//tcUNIT Common function block: Contains helper methods for tcUNIT.
FUNCTION_BLOCK FB_tcUNIT_common

VAR

END_VAR

METHOD mDisableAxis: BOOL
VAR_INPUT
    iAxisIndex: UINT; //The idex of the axis to action the method on.
END_VAR
GVL.astAxes[iAxisIndex].stControl.bEnable := FALSE;
END_METHOD

METHOD mEnableAxis: BOOL
VAR_INPUT
    iAxisIndex: UINT; //The idex of the axis to action the method on.
END_VAR
GVL.astAxes[iAxisIndex].stControl.bEnable := TRUE;
END_METHOD

METHOD mExecute: BOOL
VAR_INPUT
    iAxisIndex: UINT; //The idex of the axis to action the method on.
END_VAR
GVL.astAxes[iAxisIndex].stControl.bExecute := TRUE;
END_METHOD

METHOD mExecute_SetFALSE: BOOL
VAR_INPUT
    iAxisIndex: UINT; //The idex of the axis to action the method on.
END_VAR
GVL.astAxes[iAxisIndex].stControl.bExecute := TRUE;
END_METHOD

METHOD mGearOut : BOOL
VAR_INPUT
    iAxis: UINT;  // The idex of the axis to action the method on.
END_VAR
GVL.astAxes[iAxis].stControl.eCommand := E_MotionFunctions.eGearOut;
END_METHOD

METHOD mPrepareDefaultMove

VAR_INPUT
    iAxisIndex: UINT; //The idex of the axis to action the method on.
END_VAR
//Prepare an axis so it is ready to action a move using target defaults when executed.

GVL.astAxes[iAxisIndex].stControl.bEnable := TRUE;
GVL.astAxes[iAxisIndex].stControl.eCommand := E_MotionFunctions.eMoveAbsolute;

GVL.astAxes[iAxisIndex].stInputs.bLimitBwd := TRUE;
GVL.astAxes[iAxisIndex].stInputs.bLimitFwd := TRUE;

GVL.astAxes[iAxisIndex].stConfig.fVelocity := tcUNIT_GVL.fDEFAULT_TARGET_VELOCITY;
GVL.astAxes[iAxisIndex].stConfig.fAcceleration := tcUNIT_GVL.fDEFAULT_TARGET_ACCELERATION;
GVL.astAxes[iAxisIndex].stConfig.fDeceleration := tcUNIT_GVL.fDEFAULT_TARGET_DECCELERATION;
GVL.astAxes[iAxisIndex].stConfig.fOverride := tcUNIT_GVL.fDEFAULT_TARGET_OVERRIDE;
GVL.astAxes[iAxisIndex].stConfig.fPosition := tcUNIT_GVL.fDEFAULT_POSITION;
END_METHOD

METHOD mPrepareGearInMultiMaster
VAR_INPUT
    iAxisIndex: UINT;  // The idex of the axis to action the method on.
    astGearAxis: ARRAY[1..4] OF ST_GearAxis;
END_VAR
VAR
    i: UINT;
END_VAR
// Prepare the axis so it is ready to be coupled
GVL.astAxes[iAxisIndex].stControl.eCommand := E_MotionFunctions.eGearInMultiMaster;
FOR i:= 1 TO tcUNIT_GVL.nMAX_MASTERS DO
    GVL.astAxes[iAxisIndex].stConfig.astMultiMasterAxis[i].nIndex:=astGearAxis[i].nIndex;
    GVL.astAxes[iAxisIndex].stConfig.astMultiMasterAxis[i].fRatio:=astGearAxis[i].fRatio;
END_FOR
END_METHOD

METHOD mPrepareHome
VAR_INPUT
    iAxisIndex: UINT;  // The idex of the axis to action the method on.
    eHomingRoutine: E_HomingRoutines;
END_VAR
GVL.astAxes[iAxisIndex].stControl.eCommand := E_MotionFunctions.eHome;
GVL.astAxes[iAxisIndex].stConfig.eHomeSeq:= eHomingRoutine;
END_METHOD

METHOD mPrepareMove

VAR_INPUT
    iAxisIndex: UINT; //The idex of the axis to action the method on.
    fTargetVelocity: LREAL;
    fTargetAcceleration: LREAL;
    fTargetDeceleration: LREAL;
    fTargetPosition: LREAL;
    eMotionStrategy: E_MotionFunctions; //The desired MotionFunctions motion strategy.
END_VAR
//Prepare the axis so it is ready to action a move when executed for a given motion strategy.

GVL.astAxes[iAxisIndex].stControl.bEnable := FALSE;
GVL.astAxes[iAxisIndex].stControl.eCommand := eMotionStrategy;

GVL.astAxes[iAxisIndex].stInputs.bLimitBwd := TRUE;
GVL.astAxes[iAxisIndex].stInputs.bLimitFwd := TRUE;

GVL.astAxes[iAxisIndex].stConfig.fVelocity := fTargetVelocity;
GVL.astAxes[iAxisIndex].stConfig.fAcceleration := fTargetAcceleration;
GVL.astAxes[iAxisIndex].stConfig.fDeceleration := fTargetDeceleration;
GVL.astAxes[iAxisIndex].stConfig.fPosition := fTargetPosition;
END_METHOD

METHOD mReset : BOOL
VAR_INPUT
    iAxisIndex: UINT;  // The idex of the axis to action the method on.
END_VAR
VAR
    iCycles: UINT;
    iMaxCycles: UINT := 100;
END_VAR
GVL.astAxes[iAxisIndex].stControl.bExecute := FALSE;
FOR iCycles:= 1 TO iMaxCycles DO
    GVL.astAxes[iAxisIndex].stControl.bReset := TRUE;
    IF GVL.astaxes[iAxisIndex].stStatus.bError := FALSE THEN
        EXIT;
    END_IF
END_FOR
END_METHOD

METHOD mSetAxisDefaults

VAR_INPUT
    iAxisIndex: UINT; //The idex of the axis to action the method on.
END_VAR
// Set PLC default values for the axis. Note: Status values can take multiple cycles to updated. This is not an instant reset.

IF GVL.astAxes[iAxisIndex].stStatus.bBusy THEN
    GVL.astAxes[iAxisIndex].stControl.bStop := TRUE;
END_IF
IF GVL.astAxes[iAxisIndex].stStatus.bError THEN
    GVL.astAxes[iAxisIndex].stControl.bReset := TRUE;
END_IF
IF NOT GVL.astAxes[iAxisIndex].stControl.bEnable AND GVL.astAxes[iAxisIndex].stControl.bStop THEN
    GVL.astAxes[iAxisIndex].stControl.bStop := FALSE;
END_IF

GVL.astAxes[iAxisIndex].stControl.bEnable := FALSE;
GVL.astAxes[iAxisIndex].stControl.bExecute := FALSE;
GVL.astAxes[iAxisIndex].stControl.bReset := FALSE;
GVL.astAxes[iAxisIndex].stControl.bJogFwd := FALSE;
GVL.astAxes[iAxisIndex].stControl.bJogBwd := FALSE;
GVL.astAxes[iAxisIndex].stControl.bStop := FALSE;
GVL.astAxes[iAxisIndex].stControl.eCommand := E_MotionFunctions.eMoveAbsolute;

GVL.astAxes[iAxisIndex].stConfig.fVelocity := 0.0;
GVL.astAxes[iAxisIndex].stConfig.fAcceleration := 0.0;
GVL.astAxes[iAxisIndex].stConfig.fDeceleration := 0.0;
GVL.astAxes[iAxisIndex].stConfig.fPosition := 0;
GVL.astAxes[iAxisIndex].stConfig.fOverride := 0.0;
GVL.astAxes[iAxisIndex].stConfig.eHomeSeq := 0;

GVL.astAxes[iAxisIndex].stInputs.bLimitBwd := FALSE;
GVL.astAxes[iAxisIndex].stInputs.bLimitFwd := FALSE;
GVL.astAxes[iAxisIndex].stInputs.bHomeSensor := FALSE;
END_METHOD

END_FUNCTION_BLOCK

(* stored: Version 1.1.0.1, ProductVersion 3.1.4024.0
   POU FB_tcUNIT_common: Id {0f757d3d-99b7-46eb-bdc6-03aa126689f4}, SpecialFunc None
   Method mDisableAxis: Id {22a3dd98-69f0-4b92-8109-1b0c2fe2344d}
   Method mEnableAxis: Id {12e91532-7139-4c17-998e-4c670b584b9d}
   Method mExecute: Id {010bd927-5568-40db-a7c5-fcfe995a5cb1}
   Method mExecute_SetFALSE: Id {cc074392-b19d-414a-9010-72a4fa4d5f7a}
   Method mGearOut: Id {65c5860b-0759-45a5-a8a4-27fe9453aa76}
   Method mPrepareDefaultMove: Id {c23244d5-896c-49ad-8d8a-19390856e4dc}
   Method mPrepareGearInMultiMaster: Id {b94784af-8414-4f79-a0cd-7d3b82710c1e}
   Method mPrepareHome: Id {29a1cce2-2fc4-48e1-86f6-27b6dd699cd2}
   Method mPrepareMove: Id {97bd5417-d0a1-4d32-8732-16310a863fcc}
   Method mReset: Id {59e8bfe4-ab50-4ad3-9095-95e359837091}
   Method mSetAxisDefaults: Id {5b9336be-4414-4858-a614-0fdb2847e171} *)
